{library PUBLIC}
(* Position number type *)
TYPE PositionType : INT(1..9);
END_TYPE

(* stored: Version 1.1.0.1, ProductVersion 3.1.4024.2
   EnumerationTextList PositionType: Id {8123f690-944d-49b0-9a7f-6500d787e3a0} *)
